FUNCTION_BLOCK Service_DOControl (* Basic Function Block Type *)
  (* Standard: 61499-2 *)
  (* Version 0.0, 2014-5-4, wildai, nxtControl GmbH, Template *)
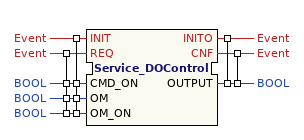
  EVENT_INPUT
    INIT WITH CMD_ON, OM, OM_ON; (* Initialization Request *)
    REQ WITH CMD_ON, OM, OM_ON; (* Normal Execution Request *)
  END_EVENT
  EVENT_OUTPUT
    INITO WITH OUTPUT; (* Initialization Confirm *)
    CNF WITH OUTPUT; (* Execution Confirmation *)
  END_EVENT
  VAR_INPUT
    CMD_ON : BOOL;
    OM : BOOL;
    OM_ON : BOOL;
  END_VAR
  VAR_OUTPUT
    OUTPUT : BOOL;
  END_VAR
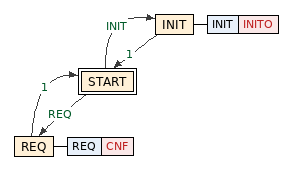
  EC_STATES
    START; (* Initial State *)
    INIT : INIT -> INITO; (* Initialization *)
    REQ : REQ -> CNF; (* Normal execution *)
  END_STATES
  EC_TRANSITIONS
    START TO INIT := INIT;
    INIT TO START := 1;
    START TO REQ := REQ;
    REQ TO START := 1;
  END_TRANSITIONS
  ALGORITHM INIT IN ST: (* Initialization algorithm *)
;
OUTPUT := FALSE;
  END_ALGORITHM
  ALGORITHM REQ IN ST: (* Normally executed algorithm *)
;

IF ((CMD_ON AND NOT OM) OR (OM AND OM_ON)) THEN
	OUTPUT := TRUE;
ELSE
	OUTPUT := FALSE;
END_IF;
  END_ALGORITHM
END_FUNCTION_BLOCK
